(* IEC 61131-3 sources: s22-soft-shell/st_interpret/tests/test_inputs/st_subset_8-9, 4 files *)

(* ---- 09_Main_Add.st ---- *)
//Testing simple function call to add two numbers together
PROGRAM 09_Main_Add
    VAR
	a : int;
        b : int;
        result0 : int;
        result1 : int;
        result2 : int;
        result3 : int;
    END_VAR
        a := 3;
        b := 5;

        // four different ways of function input
        result0 := SimpleAddFunction(10, 10+5); // expects outputs of 25

        result1 := SimpleAddFunction(Input1 := 5, Input2 := 10); // expects outputs of 15

        result2 := SimpleAddFunction(a, b); // expects outputs of 8

        result3 := SimpleAddFunction(Input1 := a, Input2 := b); // expects outputs of 8

END_PROGRAM

(* ---- 09_Main_Avg.st ---- *)
//Testing simple function call to get average of two numbers
PROGRAM 09_Main_Avg
    VAR
	a : real;
        b : real;
        avg1 : real;
        avg2 : real;
        avg3 : real;
        avg4 : real;
    END_VAR
        a := 4;
        b := 6;

        // four different ways of function input
        avg1 := ValueAverageFunction(10, 10+5); // expects 12.5

        avg2 := ValueAverageFunction(Value1 := 5, Value2 := 10); // expects 7.5

        avg3 := ValueAverageFunction(a, b); // expects 5

        avg4 := ValueAverageFunction(Value1 := a, Value2 := b); // expects 5

END_PROGRAM

(* ---- 09_Main_Context_Check.st ---- *)
//Testing to insure seperation of context, Input2 and Sum variables being used in main and add function
PROGRAM 09_Main_Context_Check
    VAR
	a : int;
        b : int;
        Input2 : int;
        Sum : INT;
        result0 : int;
        result1 : int;
    END_VAR
        a := 3;
        b := 5;
        Input2 := 10;
        Sum := 2;

        result0 := SimpleAddFunction(a, b); // expects outputs of 8

        result1 := SimpleAddFunction(Input1 := a, Input2 := b); // expects outputs of 8

END_PROGRAM

(* ---- 09_Main_Context_Check_2.st ---- *)
//Testing for calls that use the return values of two functions in the same statement
PROGRAM 09_Main_Context_Check_2
    VAR
	a : int;
        b : int;
        result0 : int;
    END_VAR
        a := 3;
        b := 5;
        result0 := 0;

        IF (SimpleAddFunction(a, b) = SimpleAddFunction(Input1 := 10, Input2 := 2) ) THEN
            result0 := 5;
        ELSEIF (SimpleAddFunction(a, b) = SimpleAddFunction(Input1 := 3, Input2 := 5) )THEN
            result0 := 10; //expected result
        ELSE
            result0 := 15;
        END_IF;

END_PROGRAM
